// TwinCAT 3 PLC project PLC1_Server
// ProgramVersion: 3.1.4024.0
// libraries:
//   Tc2_DataExchange, * (Beckhoff Automation GmbH)
//   Tc2_Standard, * (Beckhoff Automation GmbH)
//   Tc2_System, * (Beckhoff Automation GmbH)
//   Tc3_Module, * (Beckhoff Automation GmbH)
// project tree:
//   / PlcTask.TcTTO
//   POUs/ P_Server.TcPOU
// real-time tasks:
//   TASK PlcTask: cycle T#10ms, priority 20, ADS port 350
//   TASK PlcTask1: cycle T#10ms, priority 21, ADS port 351

CONFIGURATION PLC1_Server
    RESOURCE PLC ON TwinCAT3
        TASK PlcTask(INTERVAL := T#10ms, PRIORITY := 20);
        PROGRAM P_Server WITH PlcTask : P_Server;
    END_RESOURCE
END_CONFIGURATION

// ---- POUs/P_Server.TcPOU
PROGRAM P_Server
VAR
	sVar1_Read			AT%MB0		: STRING:='Beckhoff'; 	// zmienna do odczytu po adresie
	sVar1_Write			AT%MB100	: STRING;				// zmienna do zapisu po adresie
	
	sVar2_Read						: STRING:='TwinCAT';	// zmienna do odczytu po nazwie
	sVar2_Write						: STRING;				// zmienna do zapisu po nazwie 
END_VAR

;

END_PROGRAM
